Yaskawa INFORM job: TEST.JBI

/JOB
//NAME TEST
//POS
///NPOS 2,0,0,0,0,0
///TOOL 0
///POSTYPE PULSE
///PULSE
C00000=24975,-51279,139085,-4955,-130064,56275
C00001=24975,-51279,139084,-4954,-130064,56275
//INST
///DATE 2018/08/08 08:34
///ATTR SC,RW
///GROUP1 RB1
NOP
TIMER T=1.00
MOVJ C00000
MOVJ C00001 VJ=25.00
END
